Universal Robots URScript: collaborative_extension_master_52.script

######### COLLABORATIVE EXTENSION FUNCTIONS AND VARIABLES #########
global inPosSync = 0
global syncPos = [d2r(-91.71), d2r(-98.96), d2r(-126.22), d2r(-46.26), d2r(91.39), d2r(-1.78)]

tWait = 0.0005

def movel_partner(pose, a=1.2, v=0.25, t=0, r=0):

  # Wait for follower to be idle (stage 0)
  #popup("function called", "status")
  while (read_input_integer_register(25) != 0):
    sleep(tWait)
  end

  #popup("partner is idle", "status")




  # Send parameters
  write_target(pose)
  write_output_float_register(30, a)
  write_output_float_register(31, v)
  write_output_float_register(32, t)
  write_output_float_register(33, r)

  # Send command code (stage 1)
  write_output_integer_register(25, 10)

  # Wait for follower to ACK (stage 2)
  while (read_input_integer_register(25) != 2):
    sleep(tWait)
  end

  #popup("command received by partner", "status")


  # Wait for follower to finish and signal DONE (stage 3)
  while (read_input_integer_register(25) != 3):
    sleep(tWait)
  end

  #popup("partner action done", "status")


  # Reset master command register (stage 4)
  write_output_integer_register(25, 0)

  # Wait for follower to return to idle
  while (read_input_integer_register(25) != 0):
    sleep(tWait)
  end

  #popup("partner idle", "status")

end

def movej_partner(q, a=1.3, v=0.26, t=0, r=0):

  #popup("function called", "status")
  while (read_input_integer_register(25) != 0):
    sleep(tWait)
  end

  #popup("partner is idle", "status")

  write_output_integer_register(25, 11)
  write_target(q)
  write_output_float_register(30, a)
  write_output_float_register(31, v)
  write_output_float_register(32, t)
  write_output_float_register(33, r)
  # Wait for follower to ACK (stage 2)
  while (read_input_integer_register(25) != 2):
    sleep(tWait)
  end

  #popup("command received by partner", "status")

  # Wait for follower to finish and signal DONE (stage 3)
  while (read_input_integer_register(25) != 3):
    sleep(tWait)
  end

  #popup("partner action done", "status")

  # Reset master command register (stage 4)
  write_output_integer_register(25, 0)

  # Wait for follower to return to idle
  while (read_input_integer_register(25) != 0):
    sleep(tWait)
  end

  #popup("partner idle", "status")

end

def servoj_partner(q, a=0, v=0, t=0.002, lookahead_time=0.1, gain=300):
  write_output_integer_register(25, 12)
  write_target(q)
  write_output_float_register(30, a)
  write_output_float_register(31, v)
  write_output_float_register(32, t)
  write_output_float_register(33, lookahead_time)
  write_output_float_register(34, gain)
end

 def get_actual_tcp_pose_partner():
  x = read_input_float_register(38)
  y = read_input_float_register(39)
  z = read_input_float_register(40)
  rx = read_input_float_register(41)
  ry = read_input_float_register(42)
  rz = read_input_float_register(43)
  pose = p[x,y,z,rx,ry,rz]
  return pose
 end


def write_target(target):
  write_output_float_register(24, target[0])
  write_output_float_register(25, target[1])
  write_output_float_register(26, target[2])
  write_output_float_register(27, target[3])
  write_output_float_register(28, target[4])
  write_output_float_register(29, target[5])
end
######### USER PROGRAM FUNCTIONS AND VARIABLES #########

#Initialization of Variables
global programPose = p[0.079, -0.278,0.189,0.0, 3.16, 0.04]

#function and threads
def partnerThread():
 while(True):
   # popup("qNext: " + to_str(qNext), "status")
   pose = get_actual_tcp_pose()
   posePartner = get_actual_tcp_pose_partner()
   qNextPartner = get_inverse_kin(p[posePartner[0],posePartner[1],pose[2],posePartner[3],posePartner[4],posePartner[5]])
   servoj_partner(qNextPartner,0,0, 0.001,0.1, gain=1200)
 end
end

######### INITAL SYNC #########
write_output_integer_register(25, 0)

movej(syncPos, a=1.3962634015954636, v=1.0471975511965976)
movej_partner(syncPos, a=1.3962634015954636, v=1.0471975511965976)


while (True):
  programPose = p[0.079, -0.278,0.189,0.0, 3.16, 0.04]
  pose2 = programPose
  pose2[2] = pose2[2] + 0.1
  pose3 = pose2
  pose3[1] = pose3[1] + 0.1
  pose4 = pose3
  pose4[2] = pose4[2] - 0.1
  # movel_partner(programPose)
  # movel_partner(pose2)
  # movel_partner(pose3)
  # movel_partner(pose4)

  # q = syncPos
  # q1 = q + [d2r(20),d2r(0),d2r(0),d2r(0),d2r(0),d2r(0)]
  # q2 = q1 - [d2r(10),d2r(0),d2r(0),d2r(0),d2r(0),d2r(0)]
  # q3 = q2 + [d2r(10),d2r(0),d2r(0),d2r(0),d2r(0),d2r(0)]
  # q4 = q3 - [d2r(10),d2r(0),d2r(0),d2r(0),d2r(0),d2r(0)]
  # movej_partner(q, a=1.3, v=0.26, t=0, r=0)
  # movej_partner(q1, a=1.3, v=0.26, t=0, r=0)
  # movej_partner(q2, a=1.3, v=0.26, t=0, r=0)
  # movej_partner(q3, a=1.3, v=0.26, t=0, r=0)
  # movej_partner(q4, a=1.3, v=0.26, t=0, r=0)


  # movel(programPose)
  # movel_partner(programPose)
  # movel(pose2)
  # movel_partner(pose2)
  # movel(pose3)
  # movel_partner(pose3)
  # movel(pose4)
  # movel_partner(pose4)



  # movej(q, a=1.3, v=0.26, t=0, r=0)
  # movej_partner(q, a=1.3, v=0.26, t=0, r=0)
  # movej(q1, a=1.3, v=0.26, t=0, r=0)
  # movej_partner(q1, a=1.3, v=0.26, t=0, r=0)
  # movej(q2, a=1.3, v=0.26, t=0, r=0)
  # movej_partner(q2, a=1.3, v=0.26, t=0, r=0)
  # movej(q3, a=1.3, v=0.26, t=0, r=0)
  # movej_partner(q3, a=1.3, v=0.26, t=0, r=0)
  # movej(q4, a=1.3, v=0.26, t=0, r=0)
  # movej_partner(q4, a=1.3, v=0.26, t=0, r=0)

  A=0.10
  p=0
  w=2*3.1416/60 #30 is the limit but for some reson it is going twice times faster than it should in reality with w = 2pi/60 is taking 30 seconds instead of 60

  poseInit = programPose
  poseInit[0] = poseInit[0] + A
  movel(poseInit)
  movel_partner(poseInit, a=1.3, v=0.26, t=0, r=0)
  qNext = get_inverse_kin(poseInit)
  thread move_partnerThread(): partnerThread() end
  thrd = run move_partnerThread()
  while (p<=6.2831283):
    p = p + w/500
    deltaZ = A*sin(p)
    deltaX = A*cos(p)
    poseNext = p[0.079 + deltaX , -0.278, 0.189 + deltaZ ,0.0, 3.16, 0.04]
    qNext = get_inverse_kin(poseNext)
    servoj(qNext,0,0, 0.001,0.1, gain=1200)
  end
  kill thrd

end
